KUKA KRL program: MakroSubmit5.src

&ACCESS RV
&REL 10
&PARAM TEMPLATE = C:\KRC\Roboter\Template\makrosubmitvorgabe.src
&PARAM EDITMASK = MakroSubmit
&PARAM TPVW_VERSION=8.3.18
DEF MAKROSUBMIT5()
	;FOLD Makro Anfang ;%{PSE}%MKUKATPVW
	  ; interface to VW-standard routines
      EXT VW (VW_COMMAND:IN, BOOL: IN, REAL:IN, REAL:IN, REAL:IN, REAL:IN, BOOL :IN, E6POS :IN )
      RESET_MSG_DELAY (5,(CURR_SUB==5))
    ;ENDFOLD
   ; FOLD ;%{H}
END
; ENDFOLD
